Staubli VAL3: selectFile.pgx

public program selectFile(string& x_sDelimiter[], string& x_sList[])
  local num l_ni
  local num l_nj
begin
  //
  for l_nj=0 to size(x_sList)-1
    if x_sList[l_nj]!=""
      for l_ni=0 to size(x_sDelimiter)-1
        if left(x_sList[l_nj],1)==x_sDelimiter[l_ni]
          l_ni=size(x_sDelimiter)
        endIf
        if l_ni==size(x_sDelimiter)-1
          delete(x_sList[l_nj])
          l_nj=l_nj-1
        endIf
      endFor
    endIf

  endFor
end
